(* IEC 61131-3 sources: plcc/tests/fixtures/parse/error_recovery, 2 files *)

(* ---- bad_expression.st ---- *)
PROGRAM BadExpr
VAR
    x : INT;
END_VAR
    x := + * 3;
    x := 10;
END_PROGRAM

(* ---- missing_end.st ---- *)
PROGRAM Broken
VAR
    x : INT;
END_VAR
    x := 42;
